// TIA Portal V17 export
// export: Created 2024-08-09T12:53:09.9985934Z, ExportSetting WithDefaults, DisplayName Totally Integrated Automation Portal, DisplayVersion V17 Update 7, DisplayName TIA Portal Openness, DisplayVersion V17 Update 7, DisplayName TIA Portal Version Control Interface, DisplayVersion V17, DisplayName STEP 7 Professional, DisplayVersion V17 Update 7, DisplayName STEP 7 Safety, DisplayVersion V17 Update 6, DisplayName WinCC Professional, DisplayVersion V17 Update 7
VAR_GLOBAL   // PLC tag table "modulecommun"
   fgbase AT %M2000.0 : Bool;
   simul AT %M2000.1 : Bool;
   Commande_Simulation AT %MW2100 : Int;   //    {ExternalAccessible false, ExternalVisible false, ExternalWritable false}
END_VAR
VAR_GLOBAL CONSTANT   // user constants
   T_CD_EXAM : USInt := 20;
   T_LB_EXAM : USInt := 40;
   T_CD_MAT : USInt := 16;   // Longueur code matière
   T_CD_FOR : USInt := 16;   // Longueur code formule
   T_LB_FOR : USInt := 40;   // Longueur code formule
   T_LB_MAT : USInt := 40;   // Longueur libellé matière
   T_CD_VER : USInt := 16;   // Longueur version
   T_CD_REP : USInt := 16;   // Longueur répartition
   T_PROC : USInt := 20;   // Longueur nom du procédé
   T_SECT : USInt := 20;   // Longueur nom section paramauto
   T_PAR : USInt := 20;   // Longueur nom paramètre paramauto
   T_VAL : USInt := 100;   // Longueur nom valeur paramauto
   T_PACKAGE : USInt := 50;   // Longueur nom package pour contrôle version gestion
   T_FIC_LIB : USInt := 20;   // Longueur nom package pour contrôle version gestion
   NB_MAX_ORIG : USInt := 4;
   NB_MAX_DEST : SInt := 4;
   MAX_COMPO : USInt := 40;   // Nb maxi de composants
   MAX_SUB : USInt := 10;   // Nb maxi de composants de substitution
   NB_BENNES : USInt := 20;   // Nb maxi de benne de dosage
   NB_MAX_ENTBR : USInt := 5;   // Nb maxi d'entrée marche broyeur
   T_CODBAR : USInt := 80;   // Longueur code barre
   T_CD_LINC : USInt := 4;   // Longueur lieu d'incorporation
   T_ERR : USInt := 100;   // Longueur message d'erreur oracle
   T_CD_MACH : USInt := 30;   // Longueur des machines
   T_LIB_MACH : USInt := 40;   // Longueur libellé machine
   T_COMPT : USInt := 40;   // Longueur libellé compteur
   T_CD_VAL : USInt := 10;
   NB_RECUP_CEL : USInt := 20;
   T_COMM : USInt := 50;
   T_PRESENT : USInt := 16;
   T_CLIENT : USInt := 40;
   T_CD_CLIENT : USInt := 16;
   T_ADRESSE : USInt := 100;
   T_CD_POST : USInt := 10;
   T_TELEPHONE : USInt := 16;
   T_COULEUR : USInt := 16;
   T_COMMENT : USInt := 20;
   T_COMMENTAIRE : USInt := 200;
   T_CAMION : USInt := 15;
   T_IMMAT : USInt := 15;
   T_CHAUF : USInt := 50;
   T_NO_TOUR : USInt := 30;
   T_MESS : USInt := 100;   // Longueur message Vrac
   T_BOUCHE : USInt := 10;
   T_BADGE : USInt := 16;
   T_CD_OF : USInt := 20;   // Longueur code ordre de fabrication
   T_CD_DIVERS : USInt := 30;
   T_NOM_CHARG : USInt := 40;
   T_CD_DEPOT : USInt := 20;
   T_CRITERE : USInt := 20;
   T_CD_TAMIS : USInt := 20;
   NB_CB : USInt := 20;   // Nb maxi de code barre par produit
   NB_STO : USInt := 20;   // Nombre d'éléments tableau maj stock
   NB_PHASES : USInt := 10;   // Nb maxi de phases de dosage à gérer
   NB_MAX_MOBCIR : USInt := 20;
   NB_CRITERE : USInt := 5;
   T_CD_CEL : USInt := 20;
   T_CD_REC : USInt := 16;   // Longueur Code Réception (N° de commande / ERP)
   NB_DONNEES_REC : USInt := 20;   // Nombre de données max a stocker par tableau
   T_DONNEES_RE : USInt := 50;
   MAX_LOTS : USInt := 39;   // Nombre max des lots
   T_NOLOT : USInt := 20;   // Taille du numero de lot
   T_MAX_AMONTAVAL : USInt := 9;   // Taille max des taches en amont et en aval
   NB_CEL_MAX : USInt := 69;
   T_IDCOEFF_DEN : USInt := 10;   // Longeur id coeff correction densite
   Nmb_Keyword : USInt := 7;
   NB_MAX_DESTR : USInt := 19;   // Nombre max des DestR
   NB_MOB_EXT : USInt := 9;   // nombre de mobile du circuit extraction
   NB_MAX_IO : Int := 2999;
   Nbr_Max_Def : USInt := 49;
END_VAR
